// TIA Portal V19 export
DATA_BLOCK "StartStop_DB"   // DB4
// stored: InstanceOfName StartStop, InstanceOfType FB
"StartStop"
   // VAR_INPUT
   //    start : Bool;
   // END_VAR
   // VAR_OUTPUT
   //    status : Bool;
   // END_VAR
BEGIN
END_DATA_BLOCK
